FUNCTION IsGreaterThanOrEqualAnyType : BOOL
VAR_INPUT
	a					: __SYSTEM.AnyType; // A and B have to be same type
	b					: __SYSTEM.AnyType; // A and B have to be same type
END_VAR

IsGreaterThanOrEqualAnyType := NOT IsLessThanAnyType(a, b);

END_FUNCTION

(* stored: Version 1.1.0.1
   POU IsGreaterThanOrEqualAnyType: Id {e2780200-d441-0e1b-2757-946b27435d44}, SpecialFunc None *)
